{attribute 'linkalways'} 
{attribute 'no_explicit_call' := 'This FB is a CLASS and must be accessed using methods or properties'}
{attribute 'enable_dynamic_creation'}
FUNCTION_BLOCK _TcVnArray4_LREAL EXTENDS AliasDatatypeBase
VAR
	localData : TcVnArray4_LREAL;
	activeData : REFERENCE TO TcVnArray4_LREAL REF= localData;
	aliasBaseDatatype : _Array0to3OfLREAL;
END_VAR

PROPERTY PUBLIC Address : PVOID
GET
Address := ADR(activeData);
END_GET
END_PROPERTY

METHOD PUBLIC ClearReference
VAR_INPUT
END_VAR
activeData REF= localData;
SetBaseDatatypeReference();
END_METHOD

METHOD PUBLIC Clone : I_Datatype
VAR
    pClone : POINTER TO _TcVnArray4_LREAL;
END_VAR
pClone := __NEW(_TcVnArray4_LREAL);
Clone := pClone^;
END_METHOD

METHOD FB_init : BOOL
VAR_INPUT
	bInitRetains : BOOL; // if TRUE, the retain variables are initialized (warm start / cold start)
	bInCopyCode : BOOL;  // if TRUE, the instance afterwards gets moved into the copy code (online change)
	//InitialValue : TcVnArray4_LREAL; // if possible, not all values can be initialized
END_VAR
//localData := InitialValue; // if possible, not all values can be initialized
SetBaseDatatypeReference();
AddBaseDatatype(aliasBaseDatatype);
END_METHOD

PROPERTY PUBLIC Identifier : T_MAXSTRING
GET
Identifier := 'TcVnArray4_LREAL';
END_GET
END_PROPERTY

METHOD PUBLIC MakeReferenceTo
VAR_INPUT
	ReferenceTarget : REFERENCE TO TcVnArray4_LREAL;
END_VAR
activeData REF= ReferenceTarget;
SetBaseDatatypeReference();
END_METHOD

METHOD PROTECTED SetBaseDatatypeReference
VAR_INPUT
END_VAR
aliasBaseDatatype.MakeReferenceTo(activeData);
END_METHOD

PROPERTY PUBLIC Size : UDINT
GET
Size := SIZEOF(activeData);
END_GET
END_PROPERTY

METHOD TryMakeReferenceTo : BOOL
VAR_INPUT
	Target : I_Datatype;
END_VAR
VAR
	pTargetData : POINTER TO TcVnArray4_LREAL;
END_VAR
IF NOT IsEquivalentTo(Target) THEN
	RETURN;
END_IF

pTargetData := Target.Address;
activeData REF= pTargetData^;
SetBaseDatatypeReference();
TryMakeReferenceTo := TRUE;
END_METHOD

PROPERTY PUBLIC Value : REFERENCE TO TcVnArray4_LREAL
GET
Value REF= activeData;
END_GET
END_PROPERTY

END_FUNCTION_BLOCK

(* stored: Version 1.1.0.1, ProductVersion 3.1.4024.13
   POU _TcVnArray4_LREAL: Id {06cd533d-d517-08e5-13e4-c5af2db342da}, SpecialFunc None
   Folder Core: Id {777b76ea-8c6a-01aa-15c8-9c370e067625}
   Folder Protected: Id {e514576d-0077-09a5-3fd7-cb19aac962cb}
   Folder Customize: Id {489f8a64-949b-097d-1b5b-35352cfe8533}
   Folder Constructor: Id {36f3b97c-8611-0cf0-2157-21c88e2edaaf}
   Property Address: Id {42e434be-b9fa-0111-2054-cf6f5fb1d45e}
   Get Get: Id {115ec84f-444b-0199-2761-f20e3235c480}
   Method ClearReference: Id {64ad27c6-7522-0035-1a90-17a812b8246b}
   Method Clone: Id {dbf046e5-a099-0369-0e3a-a6da80870df0}
   Method FB_init: Id {b3f393c0-0812-026f-2fcb-b67ce3c50712}
   Property Identifier: Id {0cd2963a-8abb-0b02-0168-1df114a38913}
   Get Get: Id {803d6787-21ac-026c-283a-2b0c2ce955dc}
   Method MakeReferenceTo: Id {5982bd12-0c91-076c-228b-9fa03e25339a}
   Method SetBaseDatatypeReference: Id {d5b2fccc-ecd9-07d8-1bbf-9b0a042c9025}
   Property Size: Id {5db2d631-91ab-00c9-3562-5620c4cfda70}
   Get Get: Id {45e22adf-45cc-010d-04ae-411970cb9c3e}
   Method TryMakeReferenceTo: Id {6df6d9cf-6bbc-0a2a-16c7-8687d218dcbd}
   Property Value: Id {c8768e5d-3e01-0dbe-15f9-4ba4b64742fe}
   Get Get: Id {7d47ad71-7b62-0a5c-2c82-40b8deb9c8ea} *)
